{attribute 'qualified_only'}
VAR_GLOBAL
	fbAdsReturnCodes	: FB_AdsReturnCodesDescriptor;
	fbCodesysCmpErrors 	: FB_CodesysCmpErrorDescriptor;
	fbGeneralErrorCodes	: FB_GeneralCodesDescriptor;
END_VAR

(* stored: Version 1.1.0.1
   GVL GVL_ErrorDescriptors: Id {57a2c220-9d32-060d-080f-565a02024d11} *)
